FUNCTION MyFunction : T_MAXSTRING
VAR_INPUT
END_VAR
VAR
END_VAR

MyFunction := 'Hello World';

END_FUNCTION

(* stored: Version 1.1.0.1
   POU MyFunction: Id {4f0b7114-9f5e-444e-8322-38569dcddb74}, SpecialFunc None *)
